// Roboternummern:
// 
// CX-31C9D6 = 1
// CX-35CFB8 = 2
// CX-35CDC8 = 3 	!!Vorläufig
// CX-35CDD6 = 4
// CX-4D0046 = 5

VAR_GLOBAL
	Robot_Number : INT :=2;
END_VAR

(* stored: Version 1.1.0.1, ProductVersion 3.1.4026.13
   GVL Var_HAWIno: Id {fbad1c0c-79f3-465a-ba95-01cdf970df74} *)
